(* PLC project Без имени21.project, CODESYS CODESYS V3.5 SP17 Patch 3 *)
(* stored: creationDateTime 2026-04-09T19:38:53.8725276, modificationDateTime 2026-04-09T16:55:38.9994682 *)

TYPE ST_Test_Array_Init : STRUCT
  arr_int : ARRAY[1..4] OF INT := [1, 2, 3, 4];
  arr_bool : ARRAY[1..4] OF BOOL := [TRUE, FALSE, TRUE, FALSE];
END_STRUCT;
END_TYPE

TYPE ST_Test_Derived_Array_Init : STRUCT
  valve_types : ARRAY[1..3] OF INT := [1, 2, 1];
END_STRUCT;
END_TYPE

TYPE ST_Test_Map_Array_Init : STRUCT
  sensor_to_valve_map : ARRAY[1..10] OF INT := [1, 1, 1, 2, 2, 2, 2, 0, 0, 0];
END_STRUCT;
END_TYPE
